// TIA Portal V19 export
TYPE "C215_VAR_IF_DVLU_TYPIC"
   STRUCT
      STS_OPL { ExternalAccessible := 'False'; ExternalVisible := 'False'; ExternalWritable := 'False'} : Bool;   // Indicatiebord vluchtroute aangestuurd in oplopende richting
      STS_AFL { ExternalAccessible := 'False'; ExternalVisible := 'False'; ExternalWritable := 'False'} : Bool;   // Indicatiebord vluchtroute aangestuurd in aflopende richting
      EXT_AUT { ExternalAccessible := 'False'; ExternalVisible := 'False'; ExternalWritable := 'False'} : Bool;   // Externe (hoofd) beveiliging aangesproken
      EXT_HW { ExternalAccessible := 'False'; ExternalVisible := 'False'; ExternalWritable := 'False'} : Bool;   // Sturings hardware (PLC) in storing
      STO { ExternalAccessible := 'False'; ExternalVisible := 'False'; ExternalWritable := 'False'} : Struct   // Opsomming van alle storingen
         A001 : Bool;   // Beveiliging aangesproken
         AT01 : Bool;   // Foute terugmelding: Indicatiebord uitgestuurd, terugmelding Uit niet (of te laat) ontvangen
         AT02 : Bool;   // Foute terugmelding: Indicatiebord niet uitgestuurd, terugmelding Uit blijft aanwezig
         AT03 : Bool;   // Foute terugmelding: Oplopend aangestuurd, terugmelding Aan niet (of te laat) ontvangen
         AT04 : Bool;   // Foute terugmelding: Oplopend niet aangestuurd, terugmelding Aan blijft aanwezig
         AT05 : Bool;   // Foute terugmelding: Aflopend aangestuurd, terugmelding Aan niet (of te laat) ontvangen
         AT06 : Bool;   // Foute terugmelding: Aflopend niet aangestuurd, terugmelding Aan blijft aanwezig
         AT07 : Bool;   // Foute terugmeldingen: terugmeldingen oplopend en aflopend tegelijkertijd
      END_STRUCT;
   END_STRUCT;
END_TYPE
